INTERFACE PUBLIC HomingCommand EXTENDS AxisCommand

END_INTERFACE

(* stored: Version 1.1.0.1, ProductVersion 3.1.4026.13
   Itf HomingCommand: Id {c73361e5-7bfa-020c-2915-b4862cd1d4f8} *)
